// TIA Portal V17 export
// export: Created 2022-06-16T09:21:08.0839494Z, ExportSetting WithDefaults, DisplayName Totally Integrated Automation Portal, DisplayVersion V17, DisplayName TIA Portal Openness, DisplayVersion V17, DisplayName TIA Portal Version Control Interface, DisplayVersion V17, DisplayName STEP 7 Professional, DisplayVersion V17, DisplayName STEP 7 Safety, DisplayVersion V17, DisplayName WinCC Advanced, DisplayVersion V17
TYPE "typeArmGeom"
// stored: IsFailsafeCompliant false
   STRUCT
      st80Depth : Real;
      st80Offset : Real;
      st80Height : Real;
      st80Width : Real;
      st40Width : Real;
      st50Width : Real;
      outLength : Real;
      inLength : Real;
      brHeight : Real;
      st50Offset : Real;
      st80OffsetBis : Real;
      brWidth : Real;
      st80TiltOffset : Real;
   END_STRUCT;
END_TYPE
